(* PLC project Generated.project, CODESYS CODESYS V3.5 SP19 Patch 1 *)
(* stored: creationDateTime 2026-09-01T01:00:13.873199, modificationDateTime 2026-09-01T01:00:13.873199 *)

(* ═══════════════════════════════════════════════════════════════ 🎛️ ST_CycleAssistToggles — Toggles assistance mémorisés au boot 📄 Doc : DOC/AF/AF_Partie-04_Mode_SemiAuto_Sequenceur_v2.3.md §3ter ═══════════════════════════════════════════════════════════════ *)
TYPE ST_CycleAssistToggles : STRUCT
  TglEnableDiveSearch : BOOL := FALSE;  (* Mode assistance plongée mémorisé *)
  TglEnableExtractionSequence : BOOL := FALSE;  (* Mode assistance extraction mémorisé *)
  TglEnableDumpAtTremie : BOOL := FALSE;  (* Mode assistance vidage trémie mémorisé *)
  Initialized : BOOL := FALSE;  (* 🚦 flag restauration boot *)
END_STRUCT;
END_TYPE

(* ======================================================================= 💾 FB_CfgPersistBridge_CycleAssistToggles — Pont persistance toggles assistance ─────────────────────────────────────────────────────────────── 🎯 Rôle : Restauration et synchronisation bidirectionnelle IHM / Persist 💾 Persistance : Transfert GVL_PERSISTENT <-> GVL_IHM sur Initialized 📄 Doc métier : DOC/AF/AF_Partie-03_Contrats_Composants_v2.3.md §3 ======================================================================= *)
FUNCTION_BLOCK FB_CfgPersistBridge_CycleAssistToggles
  VAR_OUTPUT
    JustRestored : BOOL;  (* === ETATS RESTAURATION === <-- [STAT] Vrai sur le cycle de restauration initiale *)
  END_VAR
  VAR_IN_OUT
    Hmi : ST_CycleAssistToggles;  (* === BUS CONFIGURATION ET PERSISTANCE === <-> [BUS] Structure de toggles IHM *)
    Persist : ST_CycleAssistToggles;  (* <-> [BUS] Structure de toggles persistante *)
  END_VAR

            

JustRestored := FALSE;
IF NOT Hmi.Initialized THEN
    Hmi := Persist;
    Hmi.Initialized := TRUE;
    JustRestored := TRUE;
ELSE
    Persist := Hmi;
END_IF;

          
END_FUNCTION_BLOCK
